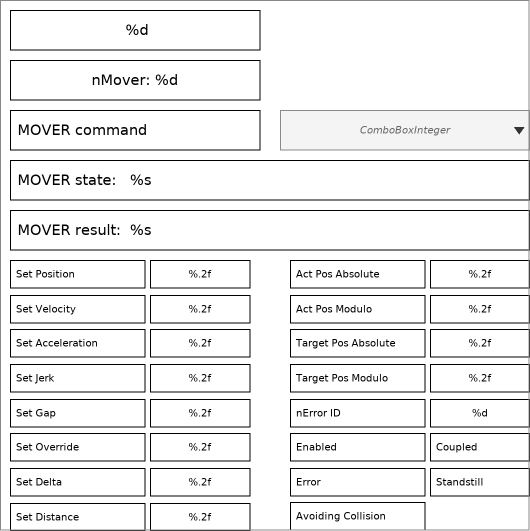
VISUALIZATION T_MOVER_SELECTOR  // 530x531
VAR_IN_OUT
	Control     : ST_MOVER_SELECTOR_CTRL;
  State       : ST_MOVER_SELECTOR_STATE;
  sState      : STRING;
  sResult     : STRING;
END_VAR
    Rectangle (10,60 250x40), "nMover: %d", text variable: Control.Mover
        OnMouseClick: write the text variable via VisuDialogs.Numpad, min 1, max MAX_MOVER, title 'Selected Mover'
    Rectangle (10,10 250x40), "%d", text variable: Control.Selector, text list: 'TL_E_MOVER_SELECTOR'
        OnMouseClick: write the text variable via VisuDialogs.Numpad, min 1, max MAX_MOVER, title 'Selected Mover'
    Rectangle (10,160 520x40), "MOVER state: %s", text variable: sState
    Rectangle (10,110 250x40), "MOVER command"
    ComboBoxInteger (280,110 250x40), variable: Control.Control.Cmd, text list: 'TL_E_CTRL_MOVER'
    Rectangle (10,210 520x40), "MOVER result: %s", text variable: sResult
    Rectangle (10,260 135x28), "Set Position"
    Rectangle (10,295 135x28), "Set Velocity"
    Rectangle (10,329 135x28), "Set Acceleration"
    Rectangle (10,364 135x28), "Set Jerk"
    Rectangle (10,399 135x28), "Set Gap"
    Rectangle (10,433 135x28), "Set Override"
    Rectangle (10,468 135x28), "Set Delta"
    Rectangle (10,503 135x28), "Set Distance"
    Rectangle (150,260 100x28), "%.2f", text variable: Control.Data.rPos
        OnMouseClick: write the text variable via Default
    Rectangle (150,295 100x28), "%.2f", text variable: Control.Data.rVelo
        OnMouseClick: write the text variable via Default
    Rectangle (150,329 100x28), "%.2f", text variable: Control.Data.rAcc
        OnMouseClick: write the text variable via Default
    Rectangle (150,364 100x28), "%.2f", text variable: Control.Data.rJerk
        OnMouseClick: write the text variable via Default
    Rectangle (150,399 100x28), "%.2f", text variable: Control.Data.rGap
        OnMouseClick: write the text variable via Default
    Rectangle (150,433 100x28), "%.2f", text variable: Control.Data.rOverride
        OnMouseClick: write the text variable via Default
    Rectangle (150,468 100x28), "%.2f", text variable: Control.Data.rDelta
        OnMouseClick: write the text variable via Default
    Rectangle (150,503 100x28), "%.2f", text variable: Control.Data.rDistance
        OnMouseClick: write the text variable via Default
    Rectangle (290,260 135x28), "Act Pos Absolute"
    Rectangle (290,295 135x28), "Act Pos Modulo"
    Rectangle (290,329 135x28), "Target Pos Absolute"
    Rectangle (290,364 135x28), "Target Pos Modulo"
    Rectangle (290,399 135x28), "nError ID"
    Rectangle (430,260 100x28), "%.2f", text variable: GVL_XTS.MoverInfo[MAIN.nMoverSelected].rAbsActPos
    Rectangle (430,295 100x28), "%.2f", text variable: GVL_XTS.MoverInfo[MAIN.nMoverSelected].rModuloActPos
    Rectangle (430,329 100x28), "%.2f", text variable: GVL_XTS.MoverInfo[MAIN.nMoverSelected].rAbsTargetPos
    Rectangle (430,364 100x28), "%.2f", text variable: GVL_XTS.MoverInfo[MAIN.nMoverSelected].rModuloTargetPos
    Rectangle (430,399 100x28), "%d", text variable: GVL_XTS.MoverInfo[MAIN.nMoverSelected].nErrorId
    Rectangle (290,433 135x28), "Enabled", colour toggle: GVL_XTS.MoverInfo[MAIN.nMoverSelected].bMoverEnabled
    Rectangle (290,468 135x28), "Error", colour toggle: GVL_XTS.MoverInfo[MAIN.nMoverSelected].bMoverError
    Rectangle (430,433 100x28), "Coupled", colour toggle: GVL_XTS.MoverInfo[MAIN.nMoverSelected].bMoverCoupled
    Rectangle (430,468 100x28), "Standstill", colour toggle: GVL_XTS.MoverInfo[MAIN.nMoverSelected].bMoverStandstill
    Rectangle (290,502 135x28), "Avoiding Collision", colour toggle: GVL_XTS.MoverInfo[MAIN.nMoverSelected].bMoverAvoidingCollision
END_VISUALIZATION

(* stored: Version 1.1.0.1, ProductVersion 3.1.4026.20
   Visu T_MOVER_SELECTOR: Id {6054c1b5-bf42-4cc5-ab26-8a7f85a9a355} *)
